TYPE DriveControl :
STRUCT
	Enable : BOOL;
	Reset : BOOL;
END_STRUCT
END_TYPE

(* stored: Version 1.1.0.1, ProductVersion 3.1.4024.9
   DUT DriveControl: Id {ee1a469a-3e1f-44b2-8855-302ff203a1e4} *)
